FUNCTION_BLOCK PtrQueue EXTENDS Queue //stores pointers to bundles, not the bundles themselves
VAR_INPUT
	
END_VAR
VAR
	elements : FB_BA_DynamicArray := (uiEntrySize := SIZEOF(PVOID), uiMinExpCount := Consts.initArraySize);
	//length : USINT := 0;
END_VAR

METHOD get : PVOID;
VAR_INPUT
	i : UINT;
END_VAR
elements.GetEntry(diIndex := i, pResultEntry := ADR(get));
END_METHOD

METHOD isEmpty : BOOL
VAR_INPUT
END_VAR
isEmpty := (elements.diCount = 0);
END_METHOD

METHOD poll : PVOID;
VAR_INST
	i : UINT;
END_VAR
poll := get(i := 0);
elements.RemoveEntry(diIndex := 0);
//length := length - 1;
END_METHOD

METHOD push : BOOL
VAR_INPUT
	value : PVOID;
END_VAR
elements.AddEntryPtr(pEntry := value);
//length := length + 1;
push := TRUE;
END_METHOD

METHOD size : DINT
VAR_INPUT
END_VAR
size := elements.diCount;
END_METHOD

END_FUNCTION_BLOCK

(* stored: Version 1.1.0.1, ProductVersion 3.1.4024.11
   POU PtrQueue: Id {2bf3e2d8-a2cd-4849-aa28-c045b8e15fa4}, SpecialFunc None
   Method get: Id {6de458e0-d05d-4d69-8bd4-22d7bdaa6891}
   Method isEmpty: Id {1ad3c8fd-cb6e-463c-88f0-72a17c67e277}
   Method poll: Id {9c526e4f-2f5b-4163-b909-8136233d5c58}
   Method push: Id {62099035-afd2-40e7-913e-ca4cb8a360e3}
   Method size: Id {6058ab76-7167-40c5-9d7b-28da77ecc464} *)
